Staubli VAL3: Glavni.pgx

program Glavni()
begin

  // pečenje samo ene palačinke

  // movej(ji,tSefla,mNomSpeed) ??

  if isSettled()
    nTaskWorking[0] = nTaskWorking[0] + 1
    call cakajProgress(1)
    call DodajMaso()
    sDiag="Peka"
    // Posodabljaj progress bar in cakaj dokler je minulu manh od nCas_peke1
    call cakajProgress(nCas_peke1)
    call obrat()
    sDiag="Peka"
    // Posodabljaj progress bar in cakaj dokler je minulu manh od nCas_peke2
    call cakajProgress(nCas_peke2)
    call naKroznik()
    // Povecaj stevec narejenih palacinke
    nCounter = nCounter + 1
    nTaskWorking[0] = nTaskWorking[0] - 1
  endIf
end
